// TIA Portal V17 export
// export: Created 2024-01-30T08:49:11.9199529Z, ExportSetting WithDefaults, DisplayName Totally Integrated Automation Portal, DisplayVersion V17 Update 6, DisplayName TIA Portal Openness, DisplayVersion V17 Update 6, DisplayName TIA Portal Version Control Interface, DisplayVersion V17, DisplayName STEP 7 Professional, DisplayVersion V17 Update 6, DisplayName STEP 7 Safety, DisplayVersion V17 Update 6, DisplayName WinCC Advanced, DisplayVersion V17 Update 6
FUNCTION_BLOCK "FB_LJ_X8000"   // FB11, LAD
{ S7_Optimized_Access := 'TRUE' }
VERSION : 0.1
// stored: AutoNumber true, IsIECCheckEnabled false, IsRetainMemResEnabled false, MemoryReserve 100, SetENOAutomatically false, UDAEnableTagReadback false
BEGIN

REGION Network 1: 02_LJ_X8000_Control
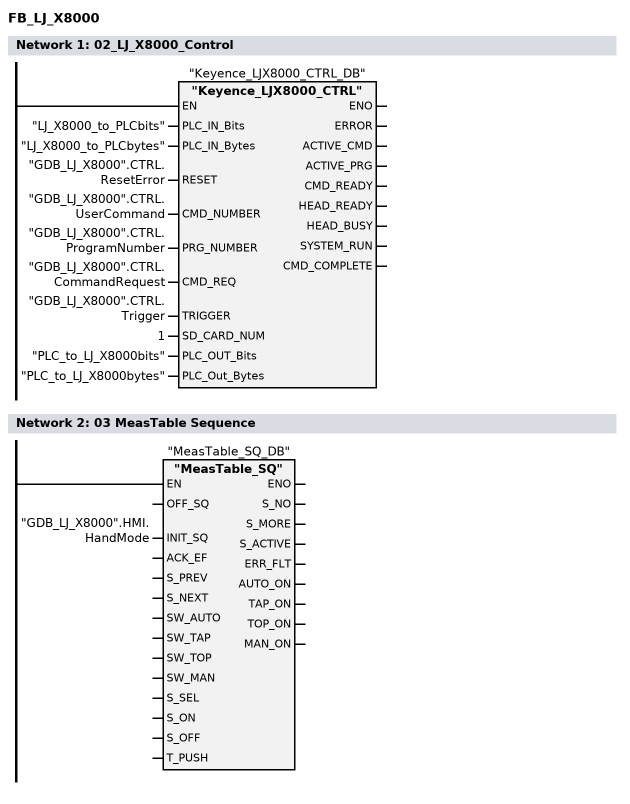
   RUNG wire#powerrail
      "Keyence_LJX8000_CTRL_DB"(PLC_IN_Bits := "LJ_X8000_to_PLCbits", PLC_IN_Bytes := "LJ_X8000_to_PLCbytes", RESET := "GDB_LJ_X8000".CTRL.ResetError, CMD_NUMBER := "GDB_LJ_X8000".CTRL.UserCommand, PRG_NUMBER := "GDB_LJ_X8000".CTRL.ProgramNumber, CMD_REQ := "GDB_LJ_X8000".CTRL.CommandRequest, TRIGGER := "GDB_LJ_X8000".CTRL.Trigger, SD_CARD_NUM := 1, PLC_OUT_Bits := "PLC_to_LJ_X8000bits", PLC_Out_Bytes := "PLC_to_LJ_X8000bytes", ERROR =>, ACTIVE_CMD =>, ACTIVE_PRG =>, CMD_READY =>, HEAD_READY =>, HEAD_BUSY =>, SYSTEM_RUN =>, CMD_COMPLETE =>)
   END_RUNG
   // the same network as SCL:
   "Keyence_LJX8000_CTRL_DB"(PLC_IN_Bits := "LJ_X8000_to_PLCbits",   // "Keyence_LJX8000_CTRL"
                           PLC_IN_Bytes := "LJ_X8000_to_PLCbytes",
                           RESET := "GDB_LJ_X8000".CTRL.ResetError,
                           CMD_NUMBER := "GDB_LJ_X8000".CTRL.UserCommand,
                           PRG_NUMBER := "GDB_LJ_X8000".CTRL.ProgramNumber,
                           CMD_REQ := "GDB_LJ_X8000".CTRL.CommandRequest,
                           TRIGGER := "GDB_LJ_X8000".CTRL.Trigger,
                           SD_CARD_NUM := 1,
                           PLC_OUT_Bits := "PLC_to_LJ_X8000bits",
                           PLC_Out_Bytes := "PLC_to_LJ_X8000bytes");
END_REGION

REGION Network 2: 03 MeasTable Sequence
   RUNG wire#powerrail
      "MeasTable_SQ_DB"(OFF_SQ :=, INIT_SQ := "GDB_LJ_X8000".HMI.HandMode, ACK_EF :=, S_PREV :=, S_NEXT :=, SW_AUTO :=, SW_TAP :=, SW_TOP :=, SW_MAN :=, S_SEL :=, S_ON :=, S_OFF :=, T_PUSH :=, S_NO =>, S_MORE =>, S_ACTIVE =>, ERR_FLT =>, AUTO_ON =>, TAP_ON =>, TOP_ON =>, MAN_ON =>)
   END_RUNG
   // the same network as SCL:
   "MeasTable_SQ_DB"(INIT_SQ := "GDB_LJ_X8000".HMI.HandMode);   // "MeasTable_SQ"
END_REGION

REGION Network 3 (SCL): 04 Battery CASE

   "MeasTable_SQ_DB".DataHasRead_1 := FALSE;

   IF "MeasTable_SQ_DB".SQ_ProgramRequest THEN

       CASE "GDB_LJ_X8000".HMI.CellType OF
           1:  // Battery cell 1
               "GDB_LJ_X8000".CTRL.ProgramNumber := 3;
               "DB_CMMT_ST".SetPosition_mm := 650.0;

           2:  // Battey cell 2 
               "GDB_LJ_X8000".CTRL.ProgramNumber := 4;
               "DB_CMMT_ST".SetPosition_mm := 712.0;
           3:  // Battery cell 3
               "GDB_LJ_X8000".CTRL.ProgramNumber := 5;
               "DB_CMMT_ST".SetPosition_mm := 815.0;
           ELSE  // Statement section ELSE
               "DB_CMMT_ST".SetPosition_mm := 240.0;
       END_CASE;

       "MeasTable_SQ_DB".DataHasRead_1 := TRUE;

   END_IF;
END_REGION

REGION Network 4 (SCL): Länge und Breite
   "GDB_LJ_X8000".Cell_MeasData.Länge := "LJ_X8000_to_PLCbytes".T101_DistanceMax / 1000.0;
   "GDB_LJ_X8000".Cell_MeasData.Breite := "LJ_X8000_to_PLCbytes".T101_NoOfNGProfiles / 1000.0;
END_REGION
END_FUNCTION_BLOCK
